(* IEC 61131-3 sources: LLHttp/, 3 files *)

(* ---- Types.typ ---- *)
(*Interface types*)

TYPE
	LLHttpHeader_typ : 	STRUCT
		contentType : STRING[LLHTTP_MAX_LEN_CONTENT_TYPE]; (*Content type *)
		contentLength : UDINT; (*Content length*)
		uri : STRING[LLHTTP_MAX_LEN_URI]; (*URI (Request)*)
		accept : STRING[LLHTTP_MAX_LEN_CONTENT_ACCEPT]; (*Content accept*)
		lines : ARRAY[0..LLHTTP_MAI_NUM_HEADER_LINES]OF LLHttpHeaderField_typ;
		version : INT; (*Http version*)
		status : INT; (*Http status (Response)*)
		method : LLHttpMethod_enum; (*Http method (Request)*)
	END_STRUCT;
	LLHttpHeaderField_typ : 	STRUCT
		name : STRING[LLHTTP_MAX_LEN_HEADER_NAME];
		value : STRING[LLHTTP_MAX_LEN_HEADER_VALUE];
	END_STRUCT;
	LLHttpMethod_enum :
		(
		LLHTTP_METHOD_GET,
		LLHTTP_METHOD_HEAD,
		LLHTTP_METHOD_POST,
		LLHTTP_METHOD_PUT,
		LLHTTP_METHOD_DELETE,
		LLHTTP_METHOD_CONNECT,
		LLHTTP_METHOD_OPTIONS,
		LLHTTP_METHOD_PATCH,
		LLHTTP_METHOD_TRACE,
		LLHTTP_METHOD_ANY, (*Match any methods*)
		LLHTTP_METHOD_DEFAULT (*Match any methods if no other matches*)
		);
	LLHttpErr_enum :
		(
		LLHTTP_ERR_VALUE_MISMATCH := -2,
		LLHTTP_ERR_NOT_FOUND := -1,
		LLHTTP_ERR_OK := 0,
		LLHTTP_ERR_PARSE := 50100,
		LLHTTP_ERR_MAX_HEADERS,
		LLHTTP_ERR_INVALID_INPUT,
		LLHTTP_ERR_PACKET_SIZE_TOO_BIG,
		LLHTTP_ERR_
		);
END_TYPE

(*Enum for the HTTP status codes.*)

TYPE
	LLHttpStatusCode_enum :
		(
		LLHTTP_STAT_Continue := 100, (* Indicates that the initial part OF a request has been received and has not yet been rejected by the server. *)
		LLHTTP_STAT_SwitchingProtocols := 101, (* Indicates that the server understands and is willing TO comply with the client's request, via the Upgrade header field, for a change in the application protocol being used on this connection. *)
		LLHTTP_STAT_Processing := 102, (* Is an interim response used TO inform the client that the server has accepted the complete request, but has not yet completed it. *)
		LLHTTP_STAT_EarlyHints := 103, (* Indicates TO the client that the server is likely TO send a final response with the header fields included in the informational response. *)
		LLHTTP_STAT_OK := 200, (* Indicates that the request has succeeded. *)
		LLHTTP_STAT_Created := 201, (* Indicates that the request has been fulfilled and has resulted in one or more new resources being created. *)
		LLHTTP_STAT_Accepted := 202, (* Indicates that the request has been accepted for processing, but the processing has not been completed. *)
		LLHTTP_STAT_NonAuthoritativeInfo := 203, (* Indicates that the request was successful but the enclosed payload has been modified from that OF the origin server's 200 (OK) response by a transforming proxy. *)
		LLHTTP_STAT_NoContent := 204, (* Indicates that the server has successfully fulfilled the request and that there is no additional content TO send in the response payload body. *)
		LLHTTP_STAT_ResetContent := 205, (* Indicates that the server has fulfilled the request and desires that the user agent reset the \"document view\", which caused the request TO be sent, to its original state as received from the origin server. *)
		LLHTTP_STAT_PartialContent := 206, (* Indicates that the server is successfully fulfilling a range request for the target resource by transferring one or more parts OF the selected representation that correspond TO the satisfiable ranges found in the requests's Range header field. *)
		LLHTTP_STAT_MultiStatus := 207, (* Provides status for multiple independent operations. *)
		LLHTTP_STAT_AlreadyReported := 208, (* Used inside a DAV:propstat response element TO avoid enumerating the internal members OF multiple bindings TO the same collection repeatedly. [RFC 5842] *)
		LLHTTP_STAT_IMUsed := 226, (* The server has fulfilled a GET request for the resource, and the response is a representation OF the result OF one or more instance-manipulations applied TO the current instance. *)
		LLHTTP_STAT_MultipleChoices := 300, (* Indicates that the target resource has more than one representation, each with its own more specific identifier, and information about the alternatives is being provided so that the user (or user agent) can select a preferred representation by redirecting its request TO one or more OF those identifiers. *)
		LLHTTP_STAT_MovedPermanently := 301, (* Indicates that the target resource has been assigned a new permanent URI and any future references TO this resource ought TO use one OF the enclosed URIs. *)
		LLHTTP_STAT_Found := 302, (* Indicates that the target resource resides temporarily under a different URI. *)
		LLHTTP_STAT_SeeOther := 303, (* Indicates that the server is redirecting the user agent TO a different resource, as indicated by a URI in the Location header field, that is intended TO provide an indirect response TO the original request. *)
		LLHTTP_STAT_NotModified := 304, (* Indicates that a conditional GET request has been received and would have resulted in a 200 (OK) response if it were not for the fact that the condition has evaluated TO false. *)
		LLHTTP_STAT_UseProxy := 305, (* \deprecated \parblock Due TO security concerns regarding in-band configuration OF a proxy. \endparblock
 The requested resource MUST be accessed through the proxy given by the Location field. *)
		LLHTTP_STAT_TemporaryRedirect := 307, (* Indicates that the target resource resides temporarily under a different URI and the user agent MUST NOT change the request method if it performs an automatic redirection TO that URI. *)
		LLHTTP_STAT_PermanentRedirect := 308, (* The target resource has been assigned a new permanent URI and any future references TO this resource ought TO use one OF the enclosed URIs. [...] This status code is similar TO 301 Moved Permanently (Section 7.3.2 OF rfc7231), except that it does not allow rewriting the request method from POST TO GET. *)
		LLHTTP_STAT_BadRequest := 400, (* Indicates that the server cannot or will not process the request because the received syntax is invalid, nonsensical, or exceeds some limitation on what the server is willing TO process. *)
		LLHTTP_STAT_Unauthorized := 401, (* Indicates that the request has not been applied because it lacks valid authentication credentials for the target resource. *)
		LLHTTP_STAT_PaymentRequired := 402, (* *Reserved* *)
		LLHTTP_STAT_Forbidden := 403, (* Indicates that the server understood the request but refuses TO authorize it. *)
		LLHTTP_STAT_NotFound := 404, (* Indicates that the origin server did not find a current representation for the target resource or is not willing TO disclose that one exists. *)
		LLHTTP_STAT_MethodNotAllowed := 405, (* Indicates that the method specified in the request-line is known by the origin server but not supported by the target resource. *)
		LLHTTP_STAT_NotAcceptable := 406, (* Indicates that the target resource does not have a current representation that would be acceptable TO the user agent, according TO the proactive negotiation header fields received in the request, and the server is unwilling TO supply a default representation. *)
		LLHTTP_STAT_ProxyAuthRequired := 407, (* Is similar TO 401 (Unauthorized), but indicates that the client needs TO authenticate itself in order TO use a proxy. *)
		LLHTTP_STAT_RequestTimeout := 408, (* Indicates that the server did not receive a complete request message within the TIME that it was prepared TO wait. *)
		LLHTTP_STAT_Conflict := 409, (* Indicates that the request could not be completed due TO a conflict with the current state OF the resource. *)
		LLHTTP_STAT_Gone := 410, (* Indicates that access TO the target resource is no longer available at the origin server and that this condition is likely TO be permanent. *)
		LLHTTP_STAT_LengthRequired := 411, (* Indicates that the server refuses TO accept the request without a defined Content-Length. *)
		LLHTTP_STAT_PreconditionFailed := 412, (* Indicates that one or more preconditions given in the request header fields evaluated TO FALSE when tested on the server. *)
		LLHTTP_STAT_PayloadTooLarge := 413, (* Indicates that the server is refusing TO process a request because the request payload is larger than the server is willing or able TO process. *)
		LLHTTP_STAT_URITooLong := 414, (* Indicates that the server is refusing TO service the request because the request-target is longer than the server is willing TO interpret. *)
		LLHTTP_STAT_UnsupportedMediaType := 415, (* Indicates that the origin server is refusing TO service the request because the payload is in a format not supported by the target resource for this method. *)
		LLHTTP_STAT_RangeNotSatisfiable := 416, (* Indicates that none OF the ranges in the request's Range header field overlap the current extent of the selected resource or that the set of ranges requested has been rejected due to invalid ranges or an excessive request of small or overlapping ranges. *)
		LLHTTP_STAT_ExpectationFailed := 417, (* Indicates that the expectation given in the request's Expect header field could not be met by at least one of the inbound servers. *)
		LLHTTP_STAT_ImATeapot := 418, (* Any attempt TO brew coffee with a teapot should result in the error code 418 I'm a teapot. *)
		LLHTTP_STAT_UnprocessableEntity := 422, (* Means the server understands the content TYPE OF the request entity (hence a 415(Unsupported Media TYPE) status code is inappropriate), and the syntax OF the request entity is correct (thus a 400 (Bad Request) status code is inappropriate) but was unable TO process the contained instructions. *)
		LLHTTP_STAT_Locked := 423, (* Means the source or destination resource OF a method is locked. *)
		LLHTTP_STAT_FailedDependency := 424, (* Means that the method could not be performed on the resource because the requested action depended on another action and that action failed. *)
		LLHTTP_STAT_UpgradeRequired := 426, (* Indicates that the server refuses TO perform the request using the current protocol but might be willing TO do so after the client upgrades TO a different protocol. *)
		LLHTTP_STAT_PreconditionRequired := 428, (* Indicates that the origin server requires the request TO be conditional. *)
		LLHTTP_STAT_TooManyRequests := 429, (* Indicates that the user has sent too many requests in a given amount OF TIME (\"rate limiting\"). *)
		LLHTTP_STAT_HeaderFieldsTooLarge := 431, (* Indicates that the server is unwilling TO process the request because its header fields are too large. *)
		LLHTTP_STAT_UnavailableLegal := 451, (* This status code indicates that the server is denying access TO the resource in response TO a legal demand. *)
		LLHTTP_STAT_InternalServerError := 500, (* Indicates that the server encountered an unexpected condition that prevented it from fulfilling the request. *)
		LLHTTP_STAT_NotImplemented := 501, (* Indicates that the server does not support the functionality required TO fulfill the request. *)
		LLHTTP_STAT_BadGateway := 502, (* Indicates that the server, while acting as a gateway or proxy, received an invalid response from an inbound server it accessed while attempting TO fulfill the request. *)
		LLHTTP_STAT_ServiceUnavailable := 503, (* Indicates that the server is currently unable TO handle the request due TO a temporary overload or scheduled maintenance, which will likely be alleviated after some delay. *)
		LLHTTP_STAT_GatewayTimeout := 504, (* Indicates that the server, while acting as a gateway or proxy, did not receive a timely response from an upstream server it needed TO access in order TO complete the request. *)
		LLHTTP_STAT_VersionNotSupported := 505, (* Indicates that the server does not support, or refuses TO support, the protocol version that was used in the request message. *)
		LLHTTP_STAT_VariantAlsoNegotiat := 506, (* Indicates that the server has an internal configuration error: the chosen variant resource is configured TO engage in transparent content negotiation itself, and is therefore not a proper end point in the negotiation process. *)
		LLHTTP_STAT_InsufficientStorage := 507, (* Means the method could not be performed on the resource because the server is unable TO store the representation needed TO successfully complete the request. *)
		LLHTTP_STAT_LoopDetected := 508, (* Indicates that the server terminated an operation because it encountered an infinite loop while processing a request with "Depth: infinity". [RFC 5842] *)
		LLHTTP_STAT_NotExtended := 510, (* The policy for accessing the resource has not been met in the request. [RFC 2774] *)
		LLHTTP_STAT_NetworkAuthRequired := 511, (* Indicates that the client needs TO authenticate TO gain network access. *)
		LLHTTP_STAT_xxx_max := 1023
		);
END_TYPE

(*Advance types*)

TYPE
	LLHttpHandler_typ : 	STRUCT
		method : LLHttpMethod_enum;
		uri : STRING[LLHTTP_MAX_LEN_URI];
		self : UDINT;
		newMessageCallback : UDINT;
		client : REFERENCE TO LLHttpServerInternalClient_typ;
		busy : BOOL;
	END_STRUCT;
	LLHttpServiceLink_typ : 	STRUCT
		requestBuffer : Buffer_typ;
		responseBuffer : Buffer_typ;
		handlers : Buffer_typ;
	END_STRUCT;
	LLHttpServiceResponse_typ : 	STRUCT
		self : UDINT;
		uri : STRING[LLHTTP_MAX_LEN_URI];
		status : UDINT;
		userHeader : ARRAY[0..LLHTTP_MAI_NUM_HEADER_LINES]OF LLHttpHeaderField_typ;
		pPayload : UDINT;
		payloadLength : UDINT;
		successCallback : UDINT;
		errorCallback : UDINT;
	END_STRUCT;
	LLHttpServiceRequest_typ : 	STRUCT
		self : UDINT;
		uri : STRING[LLHTTP_MAX_LEN_URI];
		method : UDINT;
		userHeader : ARRAY[0..LLHTTP_MAI_NUM_HEADER_LINES]OF LLHttpHeaderField_typ;
		pPayload : UDINT;
		payloadLength : UDINT;
		successCallback : UDINT;
		errorCallback : UDINT;
	END_STRUCT;
	LLHttpServerInternalClient_typ : 	STRUCT
		connected : USINT;
		tcpStream : TCPStream_typ;
		pReceiveData : {REDUND_UNREPLICABLE} UDINT;
		receiveDataSize : UDINT;
		pSendData : {REDUND_UNREPLICABLE} UDINT;
		sendDataSize : UDINT;
		sendBuffer : {REDUND_UNREPLICABLE} Buffer_typ;
		receivedBuffer : {REDUND_UNREPLICABLE} Buffer_typ;
		requestTimer : TON_10ms;
		recvLength : UDINT;
		parser : LLHttpParse;
		requestActive : BOOL;
		pCurrentRequest : REFERENCE TO LLHttpInternalRequest_typ;
		pRecvRequest : REFERENCE TO LLHttpInternalRequest_typ;
		pCurrentResponse : REFERENCE TO LLHttpServiceResponse_typ;
		api : LLHttpServiceLink_typ;
		bufferStatus : UINT;
		error : BOOL;
		errorId : DINT;
	END_STRUCT;
END_TYPE

(*Internal types*)

TYPE
	LLHttpInternalRequest_typ : 	STRUCT
		header : LLHttpHeader_typ;
		contentStart : USINT;
	END_STRUCT;
	LLHttpServerInternal_typ : 	STRUCT
		responseTimeout : TON;
		retries : UINT;
		rawrecvData : ARRAY[0..19]OF STRING[80];
		rawSendData : ARRAY[0..19]OF STRING[80];
		bufferSize : UDINT;
		tcpStream : TCPStream_typ;
		tcpMgr : TCPConnectionMgr_typ;
		bufferStatus : UDINT;
		connected : BOOL;
		state : LLHttpState_enum;
		parser : LLHttpParse;
		pClients : REFERENCE TO LLHttpServerInternalClient_typ;
		clients : ARRAY[0..LLHTTP_MAI_NUM_CLIENTS]OF LLHttpServerInternalClient_typ; (*For Debug*)
		numClientsConnected : UDINT;
		numClients : UINT;
		initialized : BOOL;
		api : LLHttpServiceLink_typ;
	END_STRUCT;
	LLHttpClientInternal_typ : 	STRUCT
		responseTimeout : TON;
		retries : UINT;
		rawrecvData : ARRAY[0..19]OF STRING[80];
		sendHeader : LLHttpHeaderField_typ;
		rawSendData : ARRAY[0..19]OF STRING[80];
		bufferSize : UDINT;
		tcpStream : TCPStream_typ;
		tcpMgr : TCPConnectionMgr_typ;
		currentRequest : LLHttpServiceRequest_typ;
		api : LLHttpServiceLink_typ;
		bufferStatus : UDINT;
		connected : BOOL;
		state : LLHttpState_enum;
		parser : LLHttpParse;
		recvLength : UDINT;
		tempBuffer : STRING[1000];
	END_STRUCT;
	LLHttpResponseInternal_typ : 	STRUCT
		send : BOOL;
		done : BOOL;
		busy : BOOL;
		error : BOOL;
		newRequest : BOOL;
		handler : LLHttpHandler_typ;
		clientApi : REFERENCE TO LLHttpServiceLink_typ;
		initialized : BOOL;
	END_STRUCT;
	LLHttpRequestInternal_typ : 	STRUCT
		send : BOOL;
		done : BOOL;
		busy : BOOL;
		error : BOOL;
	END_STRUCT;
	LLHttpState_enum :
		(
		LLHTTP_ST_IDLE,
		LLHTTP_ST_HEADER,
		LLHTTP_ST_AUTH,
		LLHTTP_ST_SEND,
		LLHTTP_ST_LISTEN,
		LLHTTP_ST_PARSE,
		LLHTTP_ST_ERROR,
		LLHTTP_ST_CLEAN,
		LLHTTP_ST_
		);
END_TYPE

(* ---- LLHttp.fun ---- *)
(*Http Usage FUBs*)

FUNCTION_BLOCK LLHttpServer (*Http Server*)
	VAR_INPUT
		enable : BOOL; (*Enable server*)
		bufferSize : UDINT; (*Size of send / recieve buffer*)
		numClients : UINT; (*Max number of clients at one time*)
		https : BOOL; (*Enable Https *)
		ipAddress : STRING[TCPCOMM_STRLEN_IPADDRESS]; (*Local IP*)
		port : UDINT; (*Local port*)
		sslIndex : UINT; (*SSl index for Https*)
	END_VAR
	VAR_OUTPUT
		ident : UDINT; (*Connection Ident*)
		numConnectedClients : UINT; (*Number of clients connected*)
		error : BOOL; (*An error occured, no acknowledge needed*)
		errorId : DINT; (*Error Id *)
	END_VAR
	VAR
		internal : LLHttpServerInternal_typ;
	END_VAR
END_FUNCTION_BLOCK

FUNCTION_BLOCK LLHttpClient (*Http Client*)
	VAR_INPUT
		enable : BOOL; (*Enable client, Client will continously try and connect to server*)
		abort : BOOL; (*Abort the existing connection*)
		bufferSize : UDINT; (*Send / Receive buffer size*)
		hostname : STRING[TCPCOMM_STRLEN_IPADDRESS]; (*Server IP or Hostname*)
		port : UINT; (*Server port (OPTIONAL)*)
		localIPAddress : STRING[TCPCOMM_STRLEN_IPADDRESS]; (*Local IP address (OPTIONAL)*)
		localPort : UINT; (*Local Port (OPTIONAL)*)
		https : BOOL; (*Use HTTPS*)
		sslIndex : UINT; (*SSL Index when using HTTPS*)
	END_VAR
	VAR_OUTPUT
		connected : BOOL; (*Connected to server *)
		ident : UDINT; (*Cient ident*)
		error : BOOL; (*An error occured, no acknowledge needed*)
		errorId : DINT;
	END_VAR
	VAR
		internal : LLHttpClientInternal_typ;
	END_VAR
END_FUNCTION_BLOCK

FUNCTION_BLOCK LLHttpRequest (*Request from header*)
	VAR_INPUT
		ident : UDINT; (*Client ident*)
		method : LLHttpMethod_enum; (*Method*)
		uri : STRING[LLHTTP_MAX_LEN_URI]; (*Host uri*)
		send : BOOL; (*Send message*)
		pUserHeader : UDINT; (*Pointer to LLHttpHeaderLine_typ array*)
		numUserHeaders : UDINT; (*Num of elements in pUserHeader*)
		pContent : UDINT; (*Body content*)
		contentType : STRING[LLHTTP_MAX_LEN_CONTENT_TYPE]; (*Content type of response content*)
		contentLength : UDINT; (*Length of content*)
		pResponse : UDINT; (*Buffer for response body*)
		responseSize : UDINT; (*Size of buffer for response body *)
	END_VAR
	VAR_OUTPUT
		header : LLHttpHeader_typ; (*Response header*)
		responseLength : UDINT; (*Response body length*)
		busy : BOOL; (*Busy, still sending or awaiting response*)
		done : BOOL; (*Request sent and response recieved *)
		error : BOOL; (*An error occured, no acknowledge needed*)
	END_VAR
	VAR
		internal : LLHttpRequestInternal_typ;
	END_VAR
END_FUNCTION_BLOCK

FUNCTION_BLOCK LLHttpResponse (*Respond to requests*)
	VAR_INPUT
		ident : UDINT; (*Client ident*)
		method : LLHttpMethod_enum; (*Request method to listen for*)
		uri : STRING[80]; (*Request URI to listen for*)
		enable : BOOL; (*Listen for requests*)
		send : BOOL; (*Send message*)
		pUserHeader : UDINT; (*Pointer to LLHttpHeaderLine_typ array*)
		numUserHeaders : UDINT; (*Num of elements in pUserHeader*)
		status : UDINT; (*Response status*)
		pContent : UDINT; (*Response body content*)
		contentType : STRING[LLHTTP_MAX_LEN_CONTENT_TYPE]; (*Content type of response content*)
		contentLength : UDINT; (*Length of response content*)
		pRequest : UDINT; (*Buffer for request body*)
		requestSize : UDINT; (*Size of buffer for request body *)
	END_VAR
	VAR_OUTPUT
		enabled : BOOL; (*Listening for requests*)
		newRequest : BOOL; (*New request recieved *)
		requestHeader : LLHttpHeader_typ; (*Response header*)
		requestLength : UDINT; (*Response body length*)
		busy : BOOL; (*Response sending*)
		done : BOOL; (*Response sent*)
		error : BOOL; (*Response error*)
	END_VAR
	VAR
		internal : {REDUND_UNREPLICABLE} LLHttpResponseInternal_typ;
	END_VAR
END_FUNCTION_BLOCK
(*Http Header evaluation*)

FUNCTION_BLOCK LLHttpParse (*Parse Http request or response*)
	VAR_INPUT
		data : UDINT; (*Pointer to data (string) to parse*)
		dataLength : UDINT; (*Length of data*)
	END_VAR
	VAR_OUTPUT
		header : LLHttpHeader_typ; (*Parsed header*)
		partialPacket : BOOL; (*Indicates partial packet*)
		partialContent : BOOL; (*Indicate partial content *)
		contentPresent : BOOL; (*Indicates content is present in message*)
		content : UDINT; (*Pointer to content*)
		error : BOOL; (*An error occured, no acknowledge needed*)
		errorId : DINT; (*Error Id*)
	END_VAR
END_FUNCTION_BLOCK

FUNCTION LLHttpHeaderContains : BOOL (*Header contains key (value?)*)
	VAR_INPUT
		headerlines : UDINT; (*Pointer to header lines*)
		name : UDINT; (*Key to find*)
		value : UDINT; (*(optional) value to find*)
	END_VAR
END_FUNCTION

FUNCTION LLHttpgetHeaderIndex : INT (*Get index of header value*)
	VAR_INPUT
		headerlines : UDINT; (*Pointer to header lines*)
		name : UDINT; (*Key to find*)
		value : UDINT; (*(optional) value to find*)
	END_VAR
END_FUNCTION

FUNCTION LLHttpAddHeaderField : DINT (*Get index of header value*)
	VAR_INPUT
		headerlines : UDINT; (*Pointer to header lines*)
		numLines : UDINT; (*Num of fields in header lines*)
		name : UDINT; (*Key to add*)
		value : UDINT; (*Value to add (optional) *)
	END_VAR
END_FUNCTION
(*Http Advance functions*)

FUNCTION LLHttpUriMatch : BOOL (*Compares two URIs*)
	VAR_INPUT
		a : UDINT; (*URI matcher, supports wildcards*)
		b : UDINT; (*URI *)
	END_VAR
END_FUNCTION

FUNCTION LLHttpMethodMatch : BOOL (*Compares two Methods*)
	VAR_INPUT
		a : LLHttpMethod_enum; (*Method 1 *)
		b : LLHttpMethod_enum; (*Method 2*)
	END_VAR
END_FUNCTION

FUNCTION LLHttpBuildResponse : DINT (*Builds response from header data*)
	VAR_INPUT
		data : UDINT; (*Buffer to be populated*)
		response : UDINT; (*LLHttpServiceResponse_typ*)
		dataSize : UDINT; (*Size of data *)
		pLen : REFERENCE TO UDINT; (*UDINT to be populated with lenght of data*)
	END_VAR
END_FUNCTION

FUNCTION LLHttpAddHandler : BOOL (*Add request handler to HTTP Server*)
	VAR_INPUT
		ident : UDINT; (*Server Ident*)
		pHandler : UDINT; (*Pointer to Handler*)
	END_VAR
END_FUNCTION
(*Http response status *)

FUNCTION LLHttpStatus_isError : BOOL (*Status is an error*)
	VAR_INPUT
		code : INT; (*Status code (HttpStatusCode_enum)*)
	END_VAR
END_FUNCTION

FUNCTION LLHttpStatus_isServerError : BOOL (*Status is a server error*)
	VAR_INPUT
		code : INT; (*Status code (HttpStatusCode_enum)*)
	END_VAR
END_FUNCTION

FUNCTION LLHttpStatus_isClientError : BOOL (*Status is a client error*)
	VAR_INPUT
		code : INT; (*Status code (HttpStatusCode_enum)*)
	END_VAR
END_FUNCTION

FUNCTION LLHttpStatus_isRedirection : BOOL (*Status is a redirect *)
	VAR_INPUT
		code : INT; (*Status code (HttpStatusCode_enum)*)
	END_VAR
END_FUNCTION

FUNCTION LLHttpStatus_isSuccessful : BOOL (*Status is success*)
	VAR_INPUT
		code : INT; (*Status code (HttpStatusCode_enum)*)
	END_VAR
END_FUNCTION

FUNCTION LLHttpStatus_isInformational : BOOL (*Status is information*)
	VAR_INPUT
		code : INT; (*Status code (HttpStatusCode_enum)*)
	END_VAR
END_FUNCTION

FUNCTION LLHttpStatus_getDescription : BOOL (*Get description from status*)
	VAR_INPUT
		code : INT; (*Status code (HttpStatusCode_enum)*)
		dest : UDINT; (*Pointer to destination to store description. Dest should be a string[24] or larger*)
	END_VAR
END_FUNCTION

(* ---- Constants.var ---- *)
VAR CONSTANT
	LLHTTP_HTTPS_PORT : UINT := 443;
	LLHTTP_HTTP_PORT : UINT := 80;
	LLHTTP_MAX_RETRIES : USINT := 5;
	LLHTTP_MAX_NUM_CLIENTS : USINT := 5;
	LLHTTP_MAI_NUM_CLIENTS : USINT := LLHTTP_MAX_NUM_CLIENTS-1;
END_VAR
(*Variable and String sizes*)
VAR CONSTANT
	LLHTTP_MAX_LEN_CONTENT_TYPE : USINT := 120;
	LLHTTP_MAX_LEN_CONTENT_ACCEPT : USINT := 255;
	LLHTTP_MAX_LEN_URI : UINT := 500;
	LLHTTP_MAX_LEN_HEADER_NAME : USINT := 120;
	LLHTTP_MAX_LEN_HEADER_VALUE : UINT := 320;
	LLHTTP_MAI_NUM_HEADER_LINES : USINT := 25;
END_VAR
